# EPICS autosave request: measCompApp/Db/C9513_chip_settings.req
$(P)$(R)FOutDivider
$(P)$(R)FOutSource
$(P)$(R)Compare1
$(P)$(R)Compare2
$(P)$(R)TimeOfDay
$(P)$(R)AlarmReg1
$(P)$(R)AlarmReg2
